TYPE U_SAFETY_MON :
UNION
	stStatusWords					: ST_SAFETY_FBStatus;		(* BUnknown, BState, wDiagnosis, wInputs, wOutputs - takie same dla wszystkich FB *)
	stStatus						: ST_SAFETY_MON; 			(* Rozbite na Bity - inne dla kazdego bloku*)
END_UNION
END_TYPE

(* stored: Version 1.1.0.1, ProductVersion 3.1.4022.12
   DUT U_SAFETY_MON: Id {e6375449-acdb-4041-aa6c-84f79e37aa2b} *)
